(*
SPDX-FileCopyrightText: © 2026 Oleksandr Tiutyk <trofimich@gmail.com>
SPDX-License-Identifier: MIT
License: https://opensource.org/license/mit
*)

(*!
<summary>Runs borrowed file-content tasks sequentially using one managed file resource.</summary>
<description>
Use one owner task; do not drive children independently while queued. DiagnosticLogger also selects the
embedded resource manager's independent diagnostic route; configure it before Start and retain its lifetime.
Child tasks retain their own diagnostic destinations. The manager owns its embedded resource
objects, not the children. Keep each child alive until removed; keep this manager alive while any child or
caller uses a borrowed resource reference. Queue removal does not clear a child's binding. Configure FilePath,
ModeFlags, PathType, AmsNetId and Timeout before Start and keep them unchanged until STOPPED. Advance Execute
through stopping and release. A completed best-effort close attempt does not prove physical close success. An
exposed handle is not an acquisition guard and must not be retained across release. Reset from STOPPED clears
queue entries and FilePath; it does not reset children. Reset in READY is a no-op. A removed STOPPED child can
Reset to clear its binding; a removed READY child must explicitly clear or replace its binding before the old
owner is destroyed. Do not mutate borrowed resource data or close its handle directly. Before online change,
stop producers from enqueueing or starting new work. For a running manager, set StopWhenNoPendingTasks to TRUE
to finish queued work, or request Cancel if abandoning waiting work is acceptable. Continue cyclic Execute
until STOPPED, including child completion and resource release. An idle running manager may still hold an open
file. Online change with a retained handle or pending native operation is unsupported; there is no automatic
guard or active-handle handoff. Cleanup errors require resolution before treating the application as prepared;
STOPPED alone does not prove physical release.
</description>
*)

{attribute 'no_explicit_call' := 'Direct call is not allowed'}
FUNCTION_BLOCK FileContentManager EXTENDS TOF_Tasks.TaskQueue
VAR_STAT
	//! <summary>Static type metadata available before the base task initializes its default name.</summary>
	{attribute 'hide'}
	_ClassName : STRING := __POUNAME();
END_VAR
VAR
	{attribute 'hide'} 
	_FileHandleResourceManager : FileHandleResourceManager;
END_VAR

(*!
<summary>Shared target for open, child operations and close. Configure before Start;</summary>
<description>
keep unchanged until STOPPED. Children obtain this target from their resource.
</description>
*)

{attribute 'monitoring' := 'call'}

PROPERTY AmsNetId : Tc2_System.T_AmsNetID
GET
AmsNetId := _FileHandleResourceManager.AmsNetId;
END_GET
SET
_FileHandleResourceManager.AmsNetId := AmsNetId;
END_SET
END_PROPERTY

(*!
<summary>Provides the concrete type name used in diagnostics.</summary>
<description>
Returns borrowed read-only metadata; keep the instance alive and do not modify the referenced string.
Initialized static storage is ready during base Task.FB_init; this getter has no side effects or exceptions.
</description>
*)
{attribute 'monitoring' := 'call'}
PROPERTY ClassName : REFERENCE TO STRING
GET
ClassName REF= _ClassName;
END_GET
END_PROPERTY

(*!
<summary>Binds a prepared file-content task to this manager and appends it to the queue.</summary>
<description>
The child is borrowed, not cloned or owned. It must be READY, alive, unique in this queue and absent from
every other queue. Do not drive or rebind it independently while queued. Successful return means the child was
appended; execution starts later through the queue. Null raises ArgumentNotSpecifiedException in the caller;
this is not a Task FAILURE result. Binding occurs before queue insertion, so an exception does not guarantee
restoration of the previous binding. A custom SetFileHandleResource may also have partial effects before
throwing. Terminal allocation failure must reach the owner's fatal task boundary. Remove a child from its
previous queue before rebinding. Removing entries does not clear their bindings. Reset this manager before
filling it for reuse from STOPPED; its Reset clears entries, not child state.
</description>
<param name="fileHandleTask">Live, unqueued READY task whose execution is delegated to this queue.</param>
*)
METHOD Enqueue
VAR_INPUT
	fileHandleTask : IFileContentTask;
END_VAR
IF fileHandleTask = 0 THEN
	(* A missing required argument cannot be reported as successful enqueue; the caller handles the exception. *)
	TOF_Core.Exceptions.ThrowArgumentNotSpecified(
		sourceNamespaceName := NamespaceName,
		sourceClassName := ClassName,
		sourcePOUName := __POUNAME(),
		sourcePosition := __POSITION(),
		argumentName := 'fileHandleTask'
	);
END_IF

fileHandleTask.SetFileHandleResource(fileHandleResource := _FileHandleResourceManager.FileHandleResource);
EnqueueTask(task := fileHandleTask);
END_METHOD

(*!
<summary>Exposes the native handle associated with this manager.</summary>
<description>
This observation does not check acquisition or physical close success. Do not close it independently or reuse
a saved value after release; file-content tasks use the manager-owned resource.
</description>
*)
{attribute 'monitoring' := 'call'}
PROPERTY FINAL FileHandle : UINT
GET
FileHandle := _FileHandleResourceManager.FileHandle;
END_GET
END_PROPERTY

{attribute 'monitoring' := 'call'}
(*!
<summary>Provides the path of the file to acquire on the configured target.</summary>
<description>
Set before Start and keep unchanged until STOPPED. The setter copies the text; the native open service
resolves it with PathType. It must refer to the target's local filesystem, not a network share. Reset from
STOPPED clears the path. Path assignment does not open or validate an existing file.
</description>
*)
PROPERTY FilePath : Tc2_System.T_MaxString
GET
FilePath := _FileHandleResourceManager.FilePath;
END_GET
SET
_FileHandleResourceManager.FilePath := FilePath;
END_SET
END_PROPERTY

(*!
<summary>Selects native file access and text or binary mode.</summary>
<description>
Configure before Start and keep unchanged until STOPPED. Choose exactly one of FOPEN_MODEREAD, FOPEN_MODEWRITE
or FOPEN_MODEAPPEND, optionally combine FOPEN_MODEPLUS, and explicitly choose one of FOPEN_MODETEXT or
FOPEN_MODEBINARY. Use Tc2_System constants with OR; incompatible choices are rejected by the native open
operation, not validated by this property. WRITE creates or truncates, READ requires an existing file, and
APPEND writes at the end. Omitting text/binary leaves the choice to the native environment. Reset preserves
these flags.
</description>
*)

{attribute 'monitoring' := 'call'}

PROPERTY ModeFlags : DWORD
GET
ModeFlags := _FileHandleResourceManager.ModeFlags;
END_GET
SET
_FileHandleResourceManager.ModeFlags := ModeFlags;
END_SET
END_PROPERTY

(*!
<summary>Provides the library namespace used in diagnostics.</summary>
<description>Returns borrowed read-only namespace storage; do not modify the referenced string.</description>
*)
{attribute 'monitoring' := 'call'}
PROPERTY NamespaceName : REFERENCE TO STRING
GET
NamespaceName REF= CurrentNamespace.Name;
END_GET
END_PROPERTY

(*!
<summary>Clears queued references and the configured file path on Reset from STOPPED.</summary>
<description>
Preserves the inherited queue reset without resetting or deleting children or clearing their resource
bindings. Other manager configuration remains unchanged. READY Reset does not invoke this hook. Overrides must
preserve both queue reset and path clearing.
</description>
*)
METHOD PROTECTED OnReset
SUPER^.OnReset();

FilePath := '';
END_METHOD

(*!
<summary>Wait for the current child and any pending file-open response before release.</summary>
<description>
Runs for every stop reason. A late handle is retained and closed by the normal resource manager.
</description>
<param name="readyToRelease">TRUE after pending work has completed and release may begin.</param>
*)

METHOD PROTECTED OnStopping
VAR_OUTPUT
	readyToRelease : BOOL;
END_VAR
SUPER^.OnStopping(readyToRelease => readyToRelease);

IF readyToRelease THEN
	readyToRelease := _FileHandleResourceManager.FinishPendingAcquire();
END_IF
END_METHOD

{attribute 'monitoring' := 'call'}
(*!
<summary>Selects the native target path context used when opening FilePath.</summary>
<description>
Configure before Start and keep unchanged until STOPPED. Passed to the native open service; it is not a
path-validity result. Reset preserves it.
</description>
*)
PROPERTY PathType : Tc2_System.E_OpenPath
GET
PathType := _FileHandleResourceManager.PathType;
END_GET
SET
_FileHandleResourceManager.PathType := PathType;
END_SET
END_PROPERTY

(*!
<summary>Exposes the file-resource manager borrowed by this task queue.</summary>
<description>
Keep this FileContentManager alive while using the interface. Use it for resource observations; do not
independently request acquisition or release, execute it, or delete it while the queue owns its lifecycle.
</description>
*)
PROPERTY ResourceManager : TOF_Core.IResourceManager
GET
ResourceManager := _FileHandleResourceManager;
END_GET
END_PROPERTY

(*!
<summary>Reports the size of this concrete instance in bytes.</summary>
*)
{attribute 'monitoring' := 'call'}
PROPERTY SelfSize : ULINT
GET
SelfSize := XSIZEOF(THIS^);
END_GET
END_PROPERTY

{attribute 'monitoring' := 'call'}
(*!
<summary>Sets the native timeout for acquiring and releasing this manager's file.</summary>
<description>
Configure before Start and keep unchanged until STOPPED. Children have their own operation timeouts; this
value is not a deadline for the whole queue or its stopping phase. Reset preserves it.
</description>
*)
PROPERTY Timeout : TIME
GET
Timeout := _FileHandleResourceManager.Timeout;
END_GET
SET
_FileHandleResourceManager.Timeout := Timeout;
END_SET
END_PROPERTY

(*!
<summary>Binds the file-resource diagnostic destination before the manager starts.</summary>
<description>
Preserves inherited start preparation. Copies the borrowed DiagnosticLogger to the embedded resource manager
without logging, I/O or ownership transfer. Keep it alive and stable through release.
</description>
*)
METHOD PROTECTED OnBeforeStart
SUPER^.OnBeforeStart();
_FileHandleResourceManager.DiagnosticLogger := THIS^.DiagnosticLogger;
END_METHOD

END_FUNCTION_BLOCK

(* stored: Version 1.1.0.1
   POU FileContentManager: Id {bc2051e9-92a1-4c8e-a38d-beb02683c33f}, SpecialFunc None
   Folder Inputs: Id {bfacd55a-3afa-44c2-84dc-abf547a00bf3}
   Folder Outputs: Id {9ba5e1c6-a771-4234-bb21-c0bdd9c29447}
   Folder Overriden members: Id {96230dd7-0bb3-48c9-8c38-e80bc28610bd}
   Property AmsNetId: Id {1c569c82-f0ee-422a-ab1a-6efc60d4b20b}
   Get Get: Id {a36a3a86-9c70-41e1-acd3-9b400a782ee7}
   Set Set: Id {5dd72bd3-ffb7-47df-9468-d7385af74eaf}
   Property ClassName: Id {7dde5df2-bee6-469e-a34d-e38f282681a9}
   Get Get: Id {d478f9e9-291b-4ed2-a175-f912be663022}
   Method Enqueue: Id {6d338e28-e90a-4f1d-be55-6a823f742ef9}
   Property FileHandle: Id {d400f36f-4560-4321-9301-560723b5321c}
   Get Get: Id {af4ff15c-e163-44de-a875-054227fd820a}
   Property FilePath: Id {f39c82db-1dee-4ac8-b085-ad0d066c8468}
   Get Get: Id {c797c652-63c0-4561-b531-110a18c85ac4}
   Set Set: Id {b19d239b-2520-4cac-89cd-a80f2163f042}
   Property ModeFlags: Id {eab34e5a-e16f-430d-90f0-029e4eb57eb1}
   Get Get: Id {cebcc8dc-c629-4eab-8dfa-12a6c42e8047}
   Set Set: Id {f58cc275-9775-4af7-bb51-396283f88ce4}
   Property NamespaceName: Id {7b18bdc5-244f-4cb6-a69d-ff82980ef6e3}
   Get Get: Id {d8cd630c-d3f9-42c5-ba22-d2cd3c67dc04}
   Method OnReset: Id {1acc0a62-c3a8-4414-bfbb-7dc3dc036945}
   Method OnStopping: Id {791680a9-1465-46a7-9d0d-334f98b2800a}
   Property PathType: Id {cbd2448b-000c-4456-acbb-370bcc431295}
   Get Get: Id {4fd9cd50-b095-453b-aa33-3b46437fbccc}
   Set Set: Id {c88e846f-0d0c-469c-b204-0549d3f33d59}
   Property ResourceManager: Id {adb82134-36e0-452b-abeb-a0acb3733da6}
   Get Get: Id {4bf105e6-40ee-4ebc-b949-d3bac16988f3}
   Property SelfSize: Id {aa575a10-da54-44bb-a1d2-ac20af742a7b}
   Get Get: Id {46726470-3c47-4383-bc77-fbfb39b4cbc0}
   Property Timeout: Id {8b8e24f2-ac37-4ffd-b14b-41645bab1c20}
   Get Get: Id {4943b545-4a96-4943-8f75-27394e4b849b}
   Set Set: Id {b3a6fe7d-0099-4655-a68b-17e02235542c}
   Method OnBeforeStart: Id {b94ab692-57fc-4f5a-9c3f-0e6bb62ec0a7} *)
